TYPE "CheckIn_ShW"
VERSION : 0.1
   STRUCT
      Trigger : Bool;
      Q_MainID : String[120];
      Q_CarrierID : Int;
      Result : Int;
      Completed : Bool;
      ProductTypeName : String[48];
      RecipeName : String[48];
      NGCode : DInt;
      ProcessCode : Int;
      TargetSubStation : Int;
      Virtual_MainID : String[48];
   END_STRUCT;

END_TYPE

